// TIA Portal V20 export
FUNCTION_BLOCK "EventsPFE"   // FB183, LAD
// stored: MemoryReserve 100, Namespace Unit1, SetENOAutomatically false
   VAR
      instResourceEvent { S7_SetPoint := 'True'} : "LPFE_ResourceEvent";
      instFEEvent_Taping { S7_SetPoint := 'True'} : "LER_LPFE_FNEvent";
      instFEEvent_HeatPressLeft { S7_SetPoint := 'True'} : "LER_LPFE_FNEvent";
      instFEEvent_HeatPressRight { S7_SetPoint := 'True'} : "LER_LPFE_FNEvent";
      instFEEvent_HipotandThickness { S7_SetPoint := 'True'} : "LER_LPFE_FNEvent";
      instFEEvent_Vision { S7_SetPoint := 'True'} : "LER_LPFE_FNEvent";
      instFEEvent_Laser { S7_SetPoint := 'True'} : "LER_LPFE_FNEvent";
      instFEEvent_Weight { S7_SetPoint := 'True'} : "LER_LPFE_FNEvent";
      InstLPFE_ValueEvent { S7_SetPoint := 'True'} : "LPFE_ValueEvent";
      InstLPFE_TelemetryEventHandlerEM0 { S7_SetPoint := 'True'} : "LPFE_TelemetryEventHandler";
      InstLPFE_TelemetryEventHandlerEM1 { S7_SetPoint := 'True'} : "LPFE_TelemetryEventHandler";
      InstLPFE_TelemetryEventHandlerEM2 { S7_SetPoint := 'True'} : "LPFE_TelemetryEventHandler";
      InstLPFE_TelemetryEventHandlerEM3 { S7_SetPoint := 'True'} : "LPFE_TelemetryEventHandler";
      InstLPFE_TelemetryEventHandlerEM4 { S7_SetPoint := 'True'} : "LPFE_TelemetryEventHandler";
      InstLPFE_TelemetryEventHandlerEM5 { S7_SetPoint := 'True'} : "LPFE_TelemetryEventHandler";
      InstLPFE_TelemetryEventHandlerEM6 { S7_SetPoint := 'True'} : "LPFE_TelemetryEventHandler";
      InstLPFE_TelemetryEventHandlerEM7 { S7_SetPoint := 'True'} : "LPFE_TelemetryEventHandler";
      InstLPFE_TelemetryEventHandlerEM8 { S7_SetPoint := 'True'} : "LPFE_TelemetryEventHandler";
      InstLPFE_TelemetryEventHandlerEM9 { S7_SetPoint := 'True'} : "LPFE_TelemetryEventHandler";
      InstLPFE_TelemetryEventHandlerEM10 { S7_SetPoint := 'True'} : "LPFE_TelemetryEventHandler";
      InstLPFE_TelemetryEventHandlerEM11 { S7_SetPoint := 'True'} : "LPFE_TelemetryEventHandler";
      InstLPFE_TelemetryEventHandlerEM12 { S7_SetPoint := 'True'} : "LPFE_TelemetryEventHandler";
      InstLPFE_TelemetryEventHandlerEM13 { S7_SetPoint := 'True'} : "LPFE_TelemetryEventHandler";
      InstLPFE_RecordEvent { S7_SetPoint := 'True'} : "LPFE_RecordEvent";
   END_VAR
BEGIN

REGION Network 1: Resource Event (4)
   // Configuration example, adpat it according to the event requirements
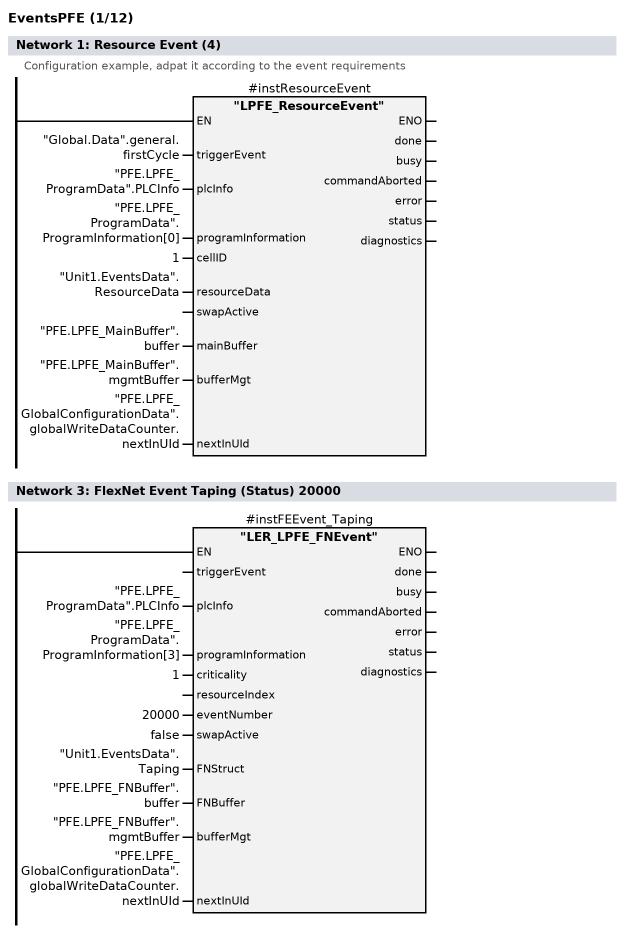
   RUNG wire#powerrail
      #instResourceEvent(triggerEvent := "Global.Data".general.firstCycle, plcInfo := "PFE.LPFE_ProgramData".PLCInfo, programInformation := "PFE.LPFE_ProgramData".ProgramInformation[0], cellID := 1, resourceData := "Unit1.EventsData".ResourceData, swapActive :=, mainBuffer := "PFE.LPFE_MainBuffer".buffer, bufferMgt := "PFE.LPFE_MainBuffer".mgmtBuffer, nextInUId := "PFE.LPFE_GlobalConfigurationData".globalWriteDataCounter.nextInUId, done =>, busy =>, commandAborted =>, error =>, status =>, diagnostics =>)
   END_RUNG
   // the same network as SCL:
   #instResourceEvent(triggerEvent := "Global.Data".general.firstCycle,   // "LPFE_ResourceEvent"
                      plcInfo := "PFE.LPFE_ProgramData".PLCInfo,
                      programInformation := "PFE.LPFE_ProgramData".ProgramInformation[0],
                      cellID := 1,
                      resourceData := "Unit1.EventsData".ResourceData,
                      mainBuffer := "PFE.LPFE_MainBuffer".buffer,
                      bufferMgt := "PFE.LPFE_MainBuffer".mgmtBuffer,
                      nextInUId := "PFE.LPFE_GlobalConfigurationData".globalWriteDataCounter.nextInUId);
END_REGION

REGION Network 3: FlexNet Event Taping (Status) 20000
   RUNG wire#powerrail
      #instFEEvent_Taping(triggerEvent :=, plcInfo := "PFE.LPFE_ProgramData".PLCInfo, programInformation := "PFE.LPFE_ProgramData".ProgramInformation[3], criticality := 1, resourceIndex :=, eventNumber := 20000, swapActive := false, FNStruct := "Unit1.EventsData".Taping, FNBuffer := "PFE.LPFE_FNBuffer".buffer, bufferMgt := "PFE.LPFE_FNBuffer".mgmtBuffer, nextInUId := "PFE.LPFE_GlobalConfigurationData".globalWriteDataCounter.nextInUId, done =>, busy =>, commandAborted =>, error =>, status =>, diagnostics =>)
   END_RUNG
   // the same network as SCL:
   #instFEEvent_Taping(plcInfo := "PFE.LPFE_ProgramData".PLCInfo,   // "LER_LPFE_FNEvent"
                       programInformation := "PFE.LPFE_ProgramData".ProgramInformation[3],
                       criticality := 1,
                       eventNumber := 20000,
                       swapActive := false,
                       FNStruct := "Unit1.EventsData".Taping,
                       FNBuffer := "PFE.LPFE_FNBuffer".buffer,
                       bufferMgt := "PFE.LPFE_FNBuffer".mgmtBuffer,
                       nextInUId := "PFE.LPFE_GlobalConfigurationData".globalWriteDataCounter.nextInUId);
END_REGION

REGION Network 4: FlexNet Event HeatPress - Left (Status) 20001
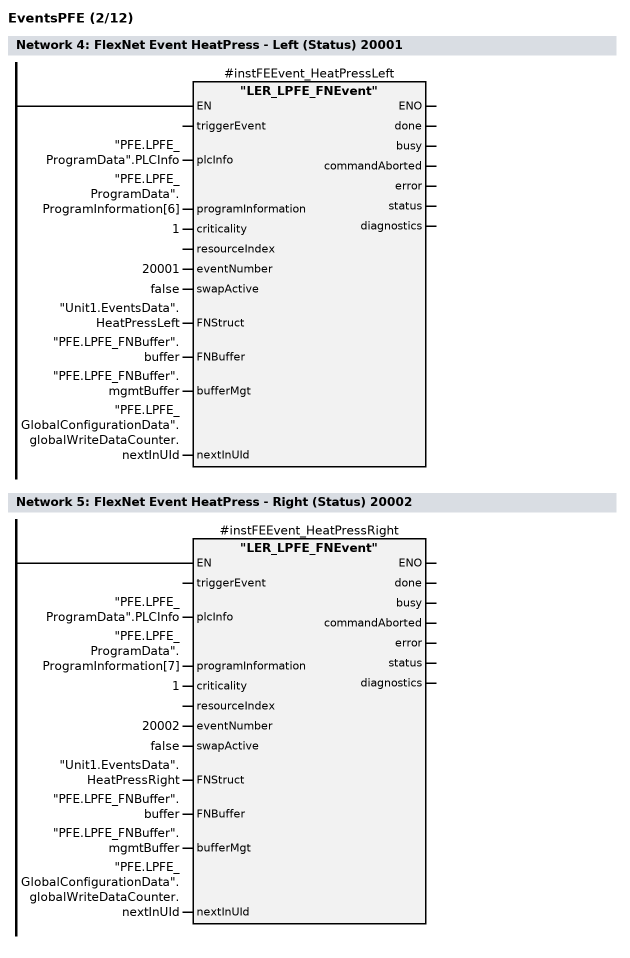
   RUNG wire#powerrail
      #instFEEvent_HeatPressLeft(triggerEvent :=, plcInfo := "PFE.LPFE_ProgramData".PLCInfo, programInformation := "PFE.LPFE_ProgramData".ProgramInformation[6], criticality := 1, resourceIndex :=, eventNumber := 20001, swapActive := false, FNStruct := "Unit1.EventsData".HeatPressLeft, FNBuffer := "PFE.LPFE_FNBuffer".buffer, bufferMgt := "PFE.LPFE_FNBuffer".mgmtBuffer, nextInUId := "PFE.LPFE_GlobalConfigurationData".globalWriteDataCounter.nextInUId, done =>, busy =>, commandAborted =>, error =>, status =>, diagnostics =>)
   END_RUNG
   // the same network as SCL:
   #instFEEvent_HeatPressLeft(plcInfo := "PFE.LPFE_ProgramData".PLCInfo,   // "LER_LPFE_FNEvent"
                           programInformation := "PFE.LPFE_ProgramData".ProgramInformation[6],
                           criticality := 1,
                           eventNumber := 20001,
                           swapActive := false,
                           FNStruct := "Unit1.EventsData".HeatPressLeft,
                           FNBuffer := "PFE.LPFE_FNBuffer".buffer,
                           bufferMgt := "PFE.LPFE_FNBuffer".mgmtBuffer,
                           nextInUId := "PFE.LPFE_GlobalConfigurationData".globalWriteDataCounter.nextInUId);
END_REGION

REGION Network 5: FlexNet Event HeatPress - Right (Status) 20002
   RUNG wire#powerrail
      #instFEEvent_HeatPressRight(triggerEvent :=, plcInfo := "PFE.LPFE_ProgramData".PLCInfo, programInformation := "PFE.LPFE_ProgramData".ProgramInformation[7], criticality := 1, resourceIndex :=, eventNumber := 20002, swapActive := false, FNStruct := "Unit1.EventsData".HeatPressRight, FNBuffer := "PFE.LPFE_FNBuffer".buffer, bufferMgt := "PFE.LPFE_FNBuffer".mgmtBuffer, nextInUId := "PFE.LPFE_GlobalConfigurationData".globalWriteDataCounter.nextInUId, done =>, busy =>, commandAborted =>, error =>, status =>, diagnostics =>)
   END_RUNG
   // the same network as SCL:
   #instFEEvent_HeatPressRight(plcInfo := "PFE.LPFE_ProgramData".PLCInfo,   // "LER_LPFE_FNEvent"
                           programInformation := "PFE.LPFE_ProgramData".ProgramInformation[7],
                           criticality := 1,
                           eventNumber := 20002,
                           swapActive := false,
                           FNStruct := "Unit1.EventsData".HeatPressRight,
                           FNBuffer := "PFE.LPFE_FNBuffer".buffer,
                           bufferMgt := "PFE.LPFE_FNBuffer".mgmtBuffer,
                           nextInUId := "PFE.LPFE_GlobalConfigurationData".globalWriteDataCounter.nextInUId);
END_REGION

REGION Network 6: FlexNet Event Hipot and Thickness (Status) 20003
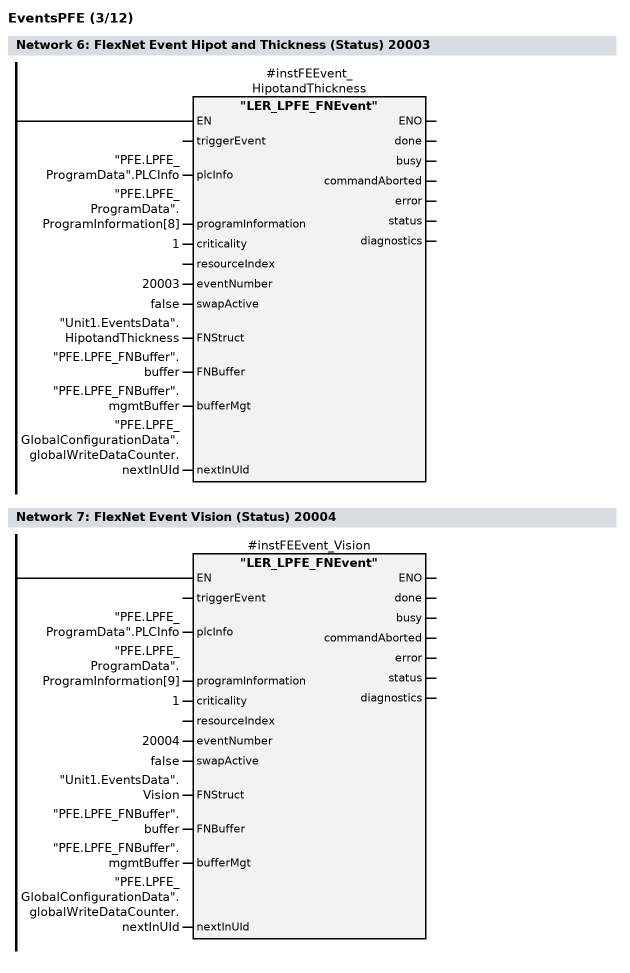
   RUNG wire#powerrail
      #instFEEvent_HipotandThickness(triggerEvent :=, plcInfo := "PFE.LPFE_ProgramData".PLCInfo, programInformation := "PFE.LPFE_ProgramData".ProgramInformation[8], criticality := 1, resourceIndex :=, eventNumber := 20003, swapActive := false, FNStruct := "Unit1.EventsData".HipotandThickness, FNBuffer := "PFE.LPFE_FNBuffer".buffer, bufferMgt := "PFE.LPFE_FNBuffer".mgmtBuffer, nextInUId := "PFE.LPFE_GlobalConfigurationData".globalWriteDataCounter.nextInUId, done =>, busy =>, commandAborted =>, error =>, status =>, diagnostics =>)
   END_RUNG
   // the same network as SCL:
   #instFEEvent_HipotandThickness(plcInfo := "PFE.LPFE_ProgramData".PLCInfo,   // "LER_LPFE_FNEvent"
                           programInformation := "PFE.LPFE_ProgramData".ProgramInformation[8],
                           criticality := 1,
                           eventNumber := 20003,
                           swapActive := false,
                           FNStruct := "Unit1.EventsData".HipotandThickness,
                           FNBuffer := "PFE.LPFE_FNBuffer".buffer,
                           bufferMgt := "PFE.LPFE_FNBuffer".mgmtBuffer,
                           nextInUId := "PFE.LPFE_GlobalConfigurationData".globalWriteDataCounter.nextInUId);
END_REGION

REGION Network 7: FlexNet Event Vision (Status) 20004
   RUNG wire#powerrail
      #instFEEvent_Vision(triggerEvent :=, plcInfo := "PFE.LPFE_ProgramData".PLCInfo, programInformation := "PFE.LPFE_ProgramData".ProgramInformation[9], criticality := 1, resourceIndex :=, eventNumber := 20004, swapActive := false, FNStruct := "Unit1.EventsData".Vision, FNBuffer := "PFE.LPFE_FNBuffer".buffer, bufferMgt := "PFE.LPFE_FNBuffer".mgmtBuffer, nextInUId := "PFE.LPFE_GlobalConfigurationData".globalWriteDataCounter.nextInUId, done =>, busy =>, commandAborted =>, error =>, status =>, diagnostics =>)
   END_RUNG
   // the same network as SCL:
   #instFEEvent_Vision(plcInfo := "PFE.LPFE_ProgramData".PLCInfo,   // "LER_LPFE_FNEvent"
                       programInformation := "PFE.LPFE_ProgramData".ProgramInformation[9],
                       criticality := 1,
                       eventNumber := 20004,
                       swapActive := false,
                       FNStruct := "Unit1.EventsData".Vision,
                       FNBuffer := "PFE.LPFE_FNBuffer".buffer,
                       bufferMgt := "PFE.LPFE_FNBuffer".mgmtBuffer,
                       nextInUId := "PFE.LPFE_GlobalConfigurationData".globalWriteDataCounter.nextInUId);
END_REGION

REGION Network 8: FlexNet Event Laser (Status) 20005
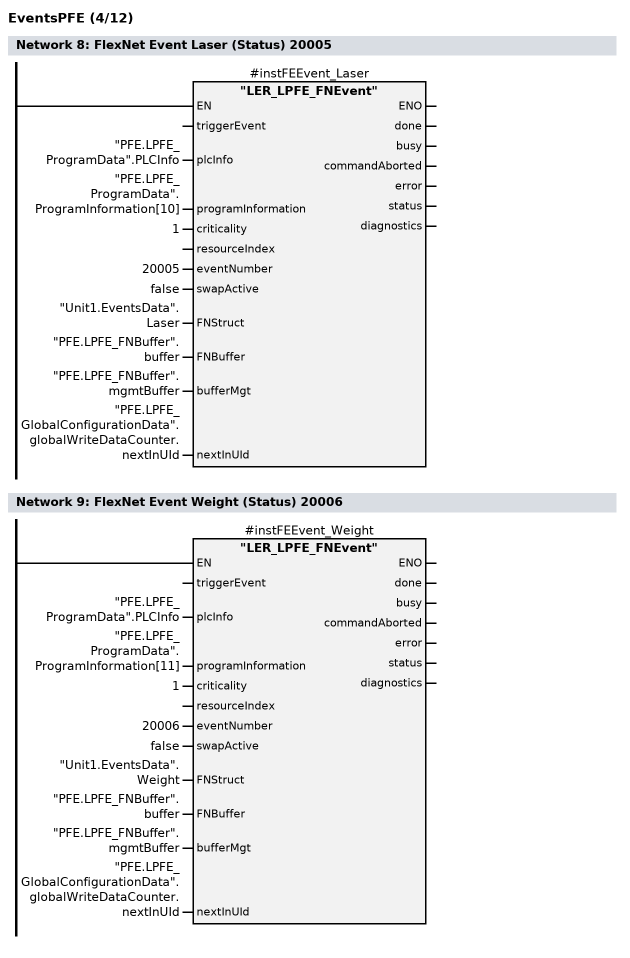
   RUNG wire#powerrail
      #instFEEvent_Laser(triggerEvent :=, plcInfo := "PFE.LPFE_ProgramData".PLCInfo, programInformation := "PFE.LPFE_ProgramData".ProgramInformation[10], criticality := 1, resourceIndex :=, eventNumber := 20005, swapActive := false, FNStruct := "Unit1.EventsData".Laser, FNBuffer := "PFE.LPFE_FNBuffer".buffer, bufferMgt := "PFE.LPFE_FNBuffer".mgmtBuffer, nextInUId := "PFE.LPFE_GlobalConfigurationData".globalWriteDataCounter.nextInUId, done =>, busy =>, commandAborted =>, error =>, status =>, diagnostics =>)
   END_RUNG
   // the same network as SCL:
   #instFEEvent_Laser(plcInfo := "PFE.LPFE_ProgramData".PLCInfo,   // "LER_LPFE_FNEvent"
                      programInformation := "PFE.LPFE_ProgramData".ProgramInformation[10],
                      criticality := 1,
                      eventNumber := 20005,
                      swapActive := false,
                      FNStruct := "Unit1.EventsData".Laser,
                      FNBuffer := "PFE.LPFE_FNBuffer".buffer,
                      bufferMgt := "PFE.LPFE_FNBuffer".mgmtBuffer,
                      nextInUId := "PFE.LPFE_GlobalConfigurationData".globalWriteDataCounter.nextInUId);
END_REGION

REGION Network 9: FlexNet Event Weight (Status) 20006
   RUNG wire#powerrail
      #instFEEvent_Weight(triggerEvent :=, plcInfo := "PFE.LPFE_ProgramData".PLCInfo, programInformation := "PFE.LPFE_ProgramData".ProgramInformation[11], criticality := 1, resourceIndex :=, eventNumber := 20006, swapActive := false, FNStruct := "Unit1.EventsData".Weight, FNBuffer := "PFE.LPFE_FNBuffer".buffer, bufferMgt := "PFE.LPFE_FNBuffer".mgmtBuffer, nextInUId := "PFE.LPFE_GlobalConfigurationData".globalWriteDataCounter.nextInUId, done =>, busy =>, commandAborted =>, error =>, status =>, diagnostics =>)
   END_RUNG
   // the same network as SCL:
   #instFEEvent_Weight(plcInfo := "PFE.LPFE_ProgramData".PLCInfo,   // "LER_LPFE_FNEvent"
                       programInformation := "PFE.LPFE_ProgramData".ProgramInformation[11],
                       criticality := 1,
                       eventNumber := 20006,
                       swapActive := false,
                       FNStruct := "Unit1.EventsData".Weight,
                       FNBuffer := "PFE.LPFE_FNBuffer".buffer,
                       bufferMgt := "PFE.LPFE_FNBuffer".mgmtBuffer,
                       nextInUId := "PFE.LPFE_GlobalConfigurationData".globalWriteDataCounter.nextInUId);
END_REGION

REGION Network 10: ValueEvent (6)
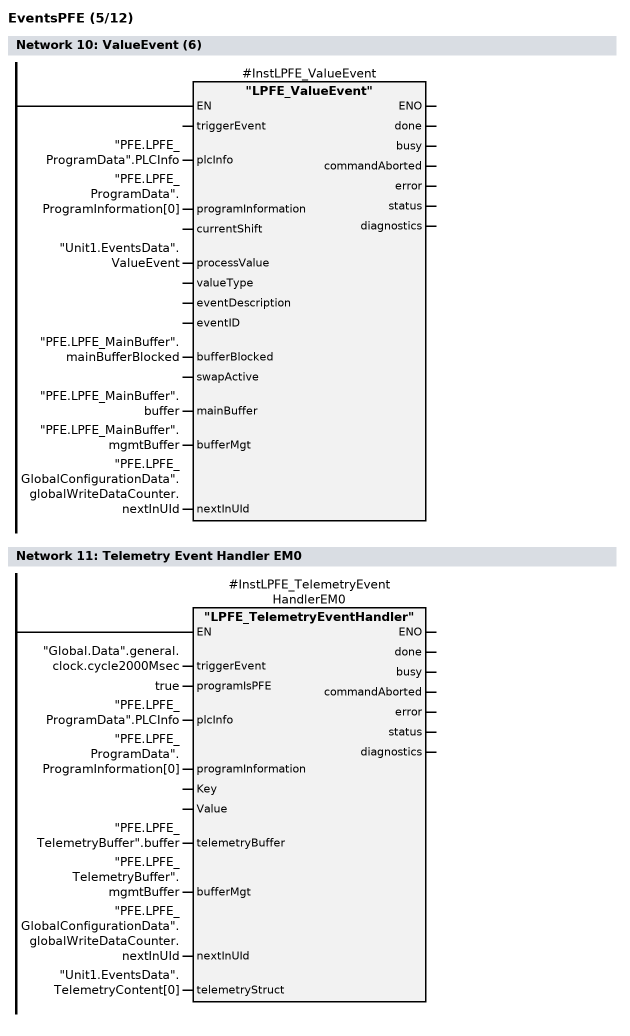
   RUNG wire#powerrail
      #InstLPFE_ValueEvent(triggerEvent :=, plcInfo := "PFE.LPFE_ProgramData".PLCInfo, programInformation := "PFE.LPFE_ProgramData".ProgramInformation[0], currentShift :=, processValue := "Unit1.EventsData".ValueEvent, valueType :=, eventDescription :=, eventID :=, bufferBlocked := "PFE.LPFE_MainBuffer".mainBufferBlocked, swapActive :=, mainBuffer := "PFE.LPFE_MainBuffer".buffer, bufferMgt := "PFE.LPFE_MainBuffer".mgmtBuffer, nextInUId := "PFE.LPFE_GlobalConfigurationData".globalWriteDataCounter.nextInUId, done =>, busy =>, commandAborted =>, error =>, status =>, diagnostics =>)
   END_RUNG
   // the same network as SCL:
   #InstLPFE_ValueEvent(plcInfo := "PFE.LPFE_ProgramData".PLCInfo,   // "LPFE_ValueEvent"
                        programInformation := "PFE.LPFE_ProgramData".ProgramInformation[0],
                        processValue := "Unit1.EventsData".ValueEvent,
                        bufferBlocked := "PFE.LPFE_MainBuffer".mainBufferBlocked,
                        mainBuffer := "PFE.LPFE_MainBuffer".buffer,
                        bufferMgt := "PFE.LPFE_MainBuffer".mgmtBuffer,
                        nextInUId := "PFE.LPFE_GlobalConfigurationData".globalWriteDataCounter.nextInUId);
END_REGION

REGION Network 11: Telemetry Event Handler EM0
   RUNG wire#powerrail
      #InstLPFE_TelemetryEventHandlerEM0(triggerEvent := "Global.Data".general.clock.cycle2000Msec, programIsPFE := true, plcInfo := "PFE.LPFE_ProgramData".PLCInfo, programInformation := "PFE.LPFE_ProgramData".ProgramInformation[0], Key :=, Value :=, telemetryBuffer := "PFE.LPFE_TelemetryBuffer".buffer, bufferMgt := "PFE.LPFE_TelemetryBuffer".mgmtBuffer, nextInUId := "PFE.LPFE_GlobalConfigurationData".globalWriteDataCounter.nextInUId, telemetryStruct := "Unit1.EventsData".TelemetryContent[0], done =>, busy =>, commandAborted =>, error =>, status =>, diagnostics =>)
   END_RUNG
   // the same network as SCL:
   #InstLPFE_TelemetryEventHandlerEM0(triggerEvent := "Global.Data".general.clock.cycle2000Msec,   // "LPFE_TelemetryEventHandler"
                           programIsPFE := true,
                           plcInfo := "PFE.LPFE_ProgramData".PLCInfo,
                           programInformation := "PFE.LPFE_ProgramData".ProgramInformation[0],
                           telemetryBuffer := "PFE.LPFE_TelemetryBuffer".buffer,
                           bufferMgt := "PFE.LPFE_TelemetryBuffer".mgmtBuffer,
                           nextInUId := "PFE.LPFE_GlobalConfigurationData".globalWriteDataCounter.nextInUId,
                           telemetryStruct := "Unit1.EventsData".TelemetryContent[0]);
END_REGION

REGION Network 12: Telemetry Event Handler EM1
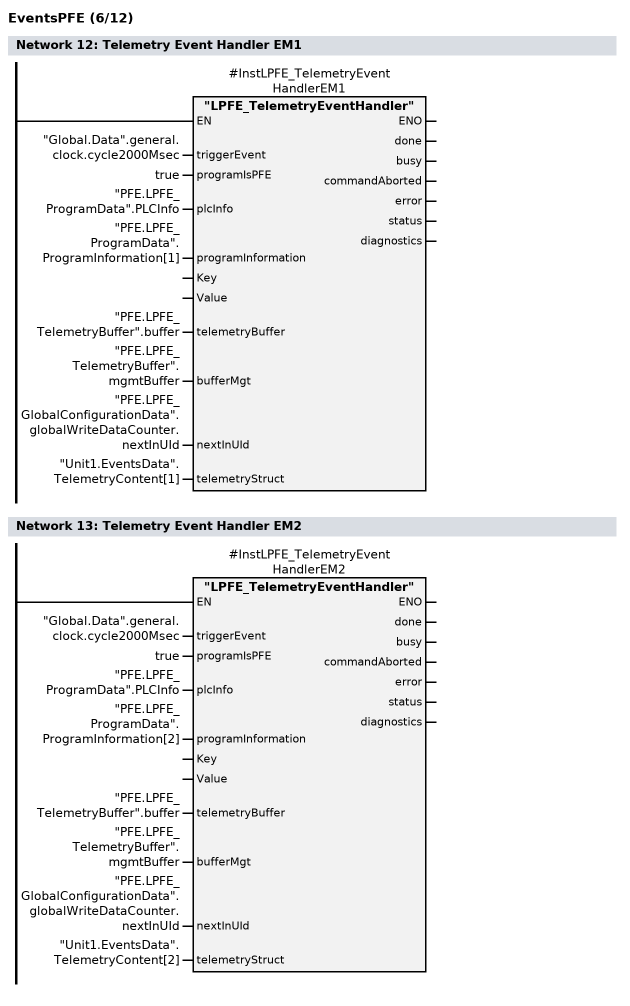
   RUNG wire#powerrail
      #InstLPFE_TelemetryEventHandlerEM1(triggerEvent := "Global.Data".general.clock.cycle2000Msec, programIsPFE := true, plcInfo := "PFE.LPFE_ProgramData".PLCInfo, programInformation := "PFE.LPFE_ProgramData".ProgramInformation[1], Key :=, Value :=, telemetryBuffer := "PFE.LPFE_TelemetryBuffer".buffer, bufferMgt := "PFE.LPFE_TelemetryBuffer".mgmtBuffer, nextInUId := "PFE.LPFE_GlobalConfigurationData".globalWriteDataCounter.nextInUId, telemetryStruct := "Unit1.EventsData".TelemetryContent[1], done =>, busy =>, commandAborted =>, error =>, status =>, diagnostics =>)
   END_RUNG
   // the same network as SCL:
   #InstLPFE_TelemetryEventHandlerEM1(triggerEvent := "Global.Data".general.clock.cycle2000Msec,   // "LPFE_TelemetryEventHandler"
                           programIsPFE := true,
                           plcInfo := "PFE.LPFE_ProgramData".PLCInfo,
                           programInformation := "PFE.LPFE_ProgramData".ProgramInformation[1],
                           telemetryBuffer := "PFE.LPFE_TelemetryBuffer".buffer,
                           bufferMgt := "PFE.LPFE_TelemetryBuffer".mgmtBuffer,
                           nextInUId := "PFE.LPFE_GlobalConfigurationData".globalWriteDataCounter.nextInUId,
                           telemetryStruct := "Unit1.EventsData".TelemetryContent[1]);
END_REGION

REGION Network 13: Telemetry Event Handler EM2
   RUNG wire#powerrail
      #InstLPFE_TelemetryEventHandlerEM2(triggerEvent := "Global.Data".general.clock.cycle2000Msec, programIsPFE := true, plcInfo := "PFE.LPFE_ProgramData".PLCInfo, programInformation := "PFE.LPFE_ProgramData".ProgramInformation[2], Key :=, Value :=, telemetryBuffer := "PFE.LPFE_TelemetryBuffer".buffer, bufferMgt := "PFE.LPFE_TelemetryBuffer".mgmtBuffer, nextInUId := "PFE.LPFE_GlobalConfigurationData".globalWriteDataCounter.nextInUId, telemetryStruct := "Unit1.EventsData".TelemetryContent[2], done =>, busy =>, commandAborted =>, error =>, status =>, diagnostics =>)
   END_RUNG
   // the same network as SCL:
   #InstLPFE_TelemetryEventHandlerEM2(triggerEvent := "Global.Data".general.clock.cycle2000Msec,   // "LPFE_TelemetryEventHandler"
                           programIsPFE := true,
                           plcInfo := "PFE.LPFE_ProgramData".PLCInfo,
                           programInformation := "PFE.LPFE_ProgramData".ProgramInformation[2],
                           telemetryBuffer := "PFE.LPFE_TelemetryBuffer".buffer,
                           bufferMgt := "PFE.LPFE_TelemetryBuffer".mgmtBuffer,
                           nextInUId := "PFE.LPFE_GlobalConfigurationData".globalWriteDataCounter.nextInUId,
                           telemetryStruct := "Unit1.EventsData".TelemetryContent[2]);
END_REGION

REGION Network 14: Telemetry Event Handler EM3
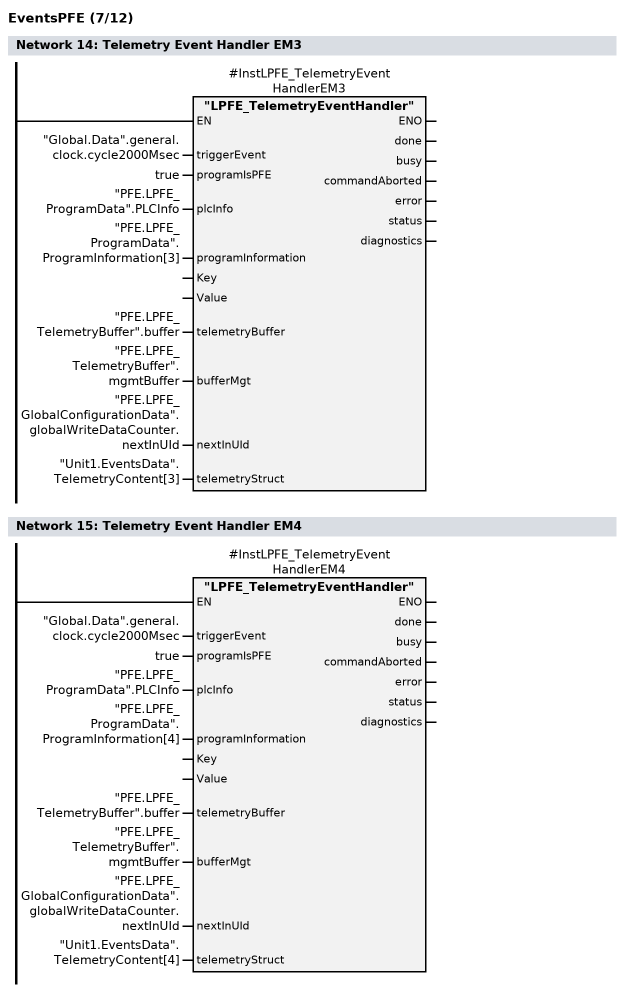
   RUNG wire#powerrail
      #InstLPFE_TelemetryEventHandlerEM3(triggerEvent := "Global.Data".general.clock.cycle2000Msec, programIsPFE := true, plcInfo := "PFE.LPFE_ProgramData".PLCInfo, programInformation := "PFE.LPFE_ProgramData".ProgramInformation[3], Key :=, Value :=, telemetryBuffer := "PFE.LPFE_TelemetryBuffer".buffer, bufferMgt := "PFE.LPFE_TelemetryBuffer".mgmtBuffer, nextInUId := "PFE.LPFE_GlobalConfigurationData".globalWriteDataCounter.nextInUId, telemetryStruct := "Unit1.EventsData".TelemetryContent[3], done =>, busy =>, commandAborted =>, error =>, status =>, diagnostics =>)
   END_RUNG
   // the same network as SCL:
   #InstLPFE_TelemetryEventHandlerEM3(triggerEvent := "Global.Data".general.clock.cycle2000Msec,   // "LPFE_TelemetryEventHandler"
                           programIsPFE := true,
                           plcInfo := "PFE.LPFE_ProgramData".PLCInfo,
                           programInformation := "PFE.LPFE_ProgramData".ProgramInformation[3],
                           telemetryBuffer := "PFE.LPFE_TelemetryBuffer".buffer,
                           bufferMgt := "PFE.LPFE_TelemetryBuffer".mgmtBuffer,
                           nextInUId := "PFE.LPFE_GlobalConfigurationData".globalWriteDataCounter.nextInUId,
                           telemetryStruct := "Unit1.EventsData".TelemetryContent[3]);
END_REGION

REGION Network 15: Telemetry Event Handler EM4
   RUNG wire#powerrail
      #InstLPFE_TelemetryEventHandlerEM4(triggerEvent := "Global.Data".general.clock.cycle2000Msec, programIsPFE := true, plcInfo := "PFE.LPFE_ProgramData".PLCInfo, programInformation := "PFE.LPFE_ProgramData".ProgramInformation[4], Key :=, Value :=, telemetryBuffer := "PFE.LPFE_TelemetryBuffer".buffer, bufferMgt := "PFE.LPFE_TelemetryBuffer".mgmtBuffer, nextInUId := "PFE.LPFE_GlobalConfigurationData".globalWriteDataCounter.nextInUId, telemetryStruct := "Unit1.EventsData".TelemetryContent[4], done =>, busy =>, commandAborted =>, error =>, status =>, diagnostics =>)
   END_RUNG
   // the same network as SCL:
   #InstLPFE_TelemetryEventHandlerEM4(triggerEvent := "Global.Data".general.clock.cycle2000Msec,   // "LPFE_TelemetryEventHandler"
                           programIsPFE := true,
                           plcInfo := "PFE.LPFE_ProgramData".PLCInfo,
                           programInformation := "PFE.LPFE_ProgramData".ProgramInformation[4],
                           telemetryBuffer := "PFE.LPFE_TelemetryBuffer".buffer,
                           bufferMgt := "PFE.LPFE_TelemetryBuffer".mgmtBuffer,
                           nextInUId := "PFE.LPFE_GlobalConfigurationData".globalWriteDataCounter.nextInUId,
                           telemetryStruct := "Unit1.EventsData".TelemetryContent[4]);
END_REGION

REGION Network 16: Telemetry Event Handler EM5
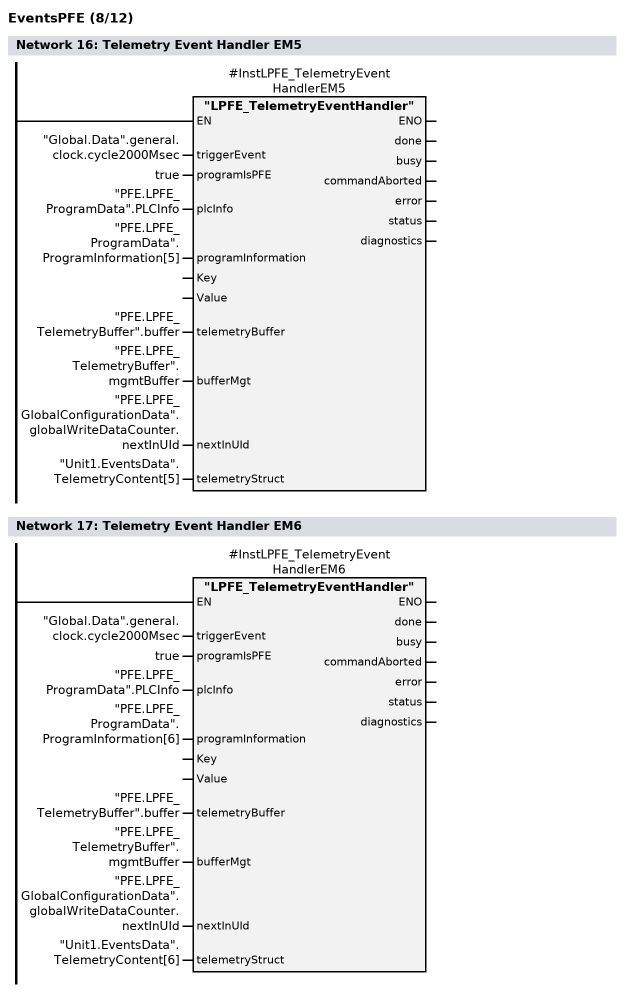
   RUNG wire#powerrail
      #InstLPFE_TelemetryEventHandlerEM5(triggerEvent := "Global.Data".general.clock.cycle2000Msec, programIsPFE := true, plcInfo := "PFE.LPFE_ProgramData".PLCInfo, programInformation := "PFE.LPFE_ProgramData".ProgramInformation[5], Key :=, Value :=, telemetryBuffer := "PFE.LPFE_TelemetryBuffer".buffer, bufferMgt := "PFE.LPFE_TelemetryBuffer".mgmtBuffer, nextInUId := "PFE.LPFE_GlobalConfigurationData".globalWriteDataCounter.nextInUId, telemetryStruct := "Unit1.EventsData".TelemetryContent[5], done =>, busy =>, commandAborted =>, error =>, status =>, diagnostics =>)
   END_RUNG
   // the same network as SCL:
   #InstLPFE_TelemetryEventHandlerEM5(triggerEvent := "Global.Data".general.clock.cycle2000Msec,   // "LPFE_TelemetryEventHandler"
                           programIsPFE := true,
                           plcInfo := "PFE.LPFE_ProgramData".PLCInfo,
                           programInformation := "PFE.LPFE_ProgramData".ProgramInformation[5],
                           telemetryBuffer := "PFE.LPFE_TelemetryBuffer".buffer,
                           bufferMgt := "PFE.LPFE_TelemetryBuffer".mgmtBuffer,
                           nextInUId := "PFE.LPFE_GlobalConfigurationData".globalWriteDataCounter.nextInUId,
                           telemetryStruct := "Unit1.EventsData".TelemetryContent[5]);
END_REGION

REGION Network 17: Telemetry Event Handler EM6
   RUNG wire#powerrail
      #InstLPFE_TelemetryEventHandlerEM6(triggerEvent := "Global.Data".general.clock.cycle2000Msec, programIsPFE := true, plcInfo := "PFE.LPFE_ProgramData".PLCInfo, programInformation := "PFE.LPFE_ProgramData".ProgramInformation[6], Key :=, Value :=, telemetryBuffer := "PFE.LPFE_TelemetryBuffer".buffer, bufferMgt := "PFE.LPFE_TelemetryBuffer".mgmtBuffer, nextInUId := "PFE.LPFE_GlobalConfigurationData".globalWriteDataCounter.nextInUId, telemetryStruct := "Unit1.EventsData".TelemetryContent[6], done =>, busy =>, commandAborted =>, error =>, status =>, diagnostics =>)
   END_RUNG
   // the same network as SCL:
   #InstLPFE_TelemetryEventHandlerEM6(triggerEvent := "Global.Data".general.clock.cycle2000Msec,   // "LPFE_TelemetryEventHandler"
                           programIsPFE := true,
                           plcInfo := "PFE.LPFE_ProgramData".PLCInfo,
                           programInformation := "PFE.LPFE_ProgramData".ProgramInformation[6],
                           telemetryBuffer := "PFE.LPFE_TelemetryBuffer".buffer,
                           bufferMgt := "PFE.LPFE_TelemetryBuffer".mgmtBuffer,
                           nextInUId := "PFE.LPFE_GlobalConfigurationData".globalWriteDataCounter.nextInUId,
                           telemetryStruct := "Unit1.EventsData".TelemetryContent[6]);
END_REGION

REGION Network 18: Telemetry Event Handler EM7
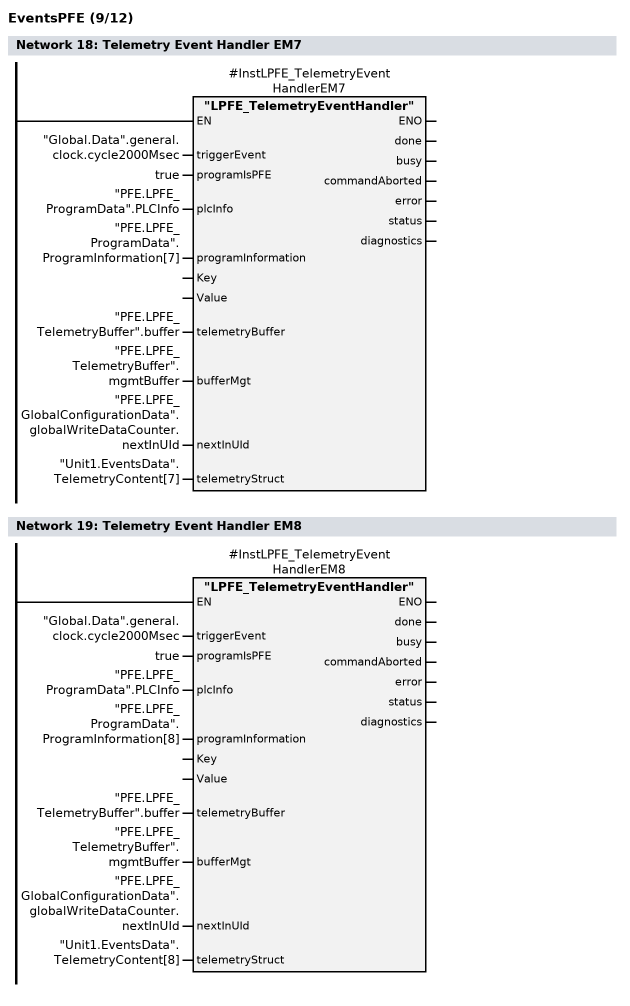
   RUNG wire#powerrail
      #InstLPFE_TelemetryEventHandlerEM7(triggerEvent := "Global.Data".general.clock.cycle2000Msec, programIsPFE := true, plcInfo := "PFE.LPFE_ProgramData".PLCInfo, programInformation := "PFE.LPFE_ProgramData".ProgramInformation[7], Key :=, Value :=, telemetryBuffer := "PFE.LPFE_TelemetryBuffer".buffer, bufferMgt := "PFE.LPFE_TelemetryBuffer".mgmtBuffer, nextInUId := "PFE.LPFE_GlobalConfigurationData".globalWriteDataCounter.nextInUId, telemetryStruct := "Unit1.EventsData".TelemetryContent[7], done =>, busy =>, commandAborted =>, error =>, status =>, diagnostics =>)
   END_RUNG
   // the same network as SCL:
   #InstLPFE_TelemetryEventHandlerEM7(triggerEvent := "Global.Data".general.clock.cycle2000Msec,   // "LPFE_TelemetryEventHandler"
                           programIsPFE := true,
                           plcInfo := "PFE.LPFE_ProgramData".PLCInfo,
                           programInformation := "PFE.LPFE_ProgramData".ProgramInformation[7],
                           telemetryBuffer := "PFE.LPFE_TelemetryBuffer".buffer,
                           bufferMgt := "PFE.LPFE_TelemetryBuffer".mgmtBuffer,
                           nextInUId := "PFE.LPFE_GlobalConfigurationData".globalWriteDataCounter.nextInUId,
                           telemetryStruct := "Unit1.EventsData".TelemetryContent[7]);
END_REGION

REGION Network 19: Telemetry Event Handler EM8
   RUNG wire#powerrail
      #InstLPFE_TelemetryEventHandlerEM8(triggerEvent := "Global.Data".general.clock.cycle2000Msec, programIsPFE := true, plcInfo := "PFE.LPFE_ProgramData".PLCInfo, programInformation := "PFE.LPFE_ProgramData".ProgramInformation[8], Key :=, Value :=, telemetryBuffer := "PFE.LPFE_TelemetryBuffer".buffer, bufferMgt := "PFE.LPFE_TelemetryBuffer".mgmtBuffer, nextInUId := "PFE.LPFE_GlobalConfigurationData".globalWriteDataCounter.nextInUId, telemetryStruct := "Unit1.EventsData".TelemetryContent[8], done =>, busy =>, commandAborted =>, error =>, status =>, diagnostics =>)
   END_RUNG
   // the same network as SCL:
   #InstLPFE_TelemetryEventHandlerEM8(triggerEvent := "Global.Data".general.clock.cycle2000Msec,   // "LPFE_TelemetryEventHandler"
                           programIsPFE := true,
                           plcInfo := "PFE.LPFE_ProgramData".PLCInfo,
                           programInformation := "PFE.LPFE_ProgramData".ProgramInformation[8],
                           telemetryBuffer := "PFE.LPFE_TelemetryBuffer".buffer,
                           bufferMgt := "PFE.LPFE_TelemetryBuffer".mgmtBuffer,
                           nextInUId := "PFE.LPFE_GlobalConfigurationData".globalWriteDataCounter.nextInUId,
                           telemetryStruct := "Unit1.EventsData".TelemetryContent[8]);
END_REGION

REGION Network 20: Telemetry Event Handler EM9
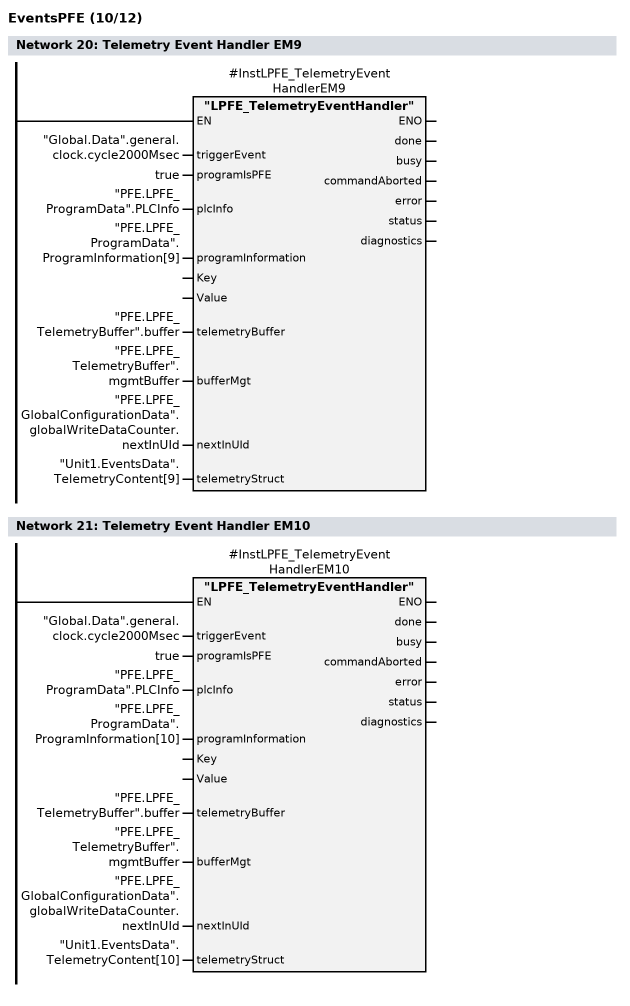
   RUNG wire#powerrail
      #InstLPFE_TelemetryEventHandlerEM9(triggerEvent := "Global.Data".general.clock.cycle2000Msec, programIsPFE := true, plcInfo := "PFE.LPFE_ProgramData".PLCInfo, programInformation := "PFE.LPFE_ProgramData".ProgramInformation[9], Key :=, Value :=, telemetryBuffer := "PFE.LPFE_TelemetryBuffer".buffer, bufferMgt := "PFE.LPFE_TelemetryBuffer".mgmtBuffer, nextInUId := "PFE.LPFE_GlobalConfigurationData".globalWriteDataCounter.nextInUId, telemetryStruct := "Unit1.EventsData".TelemetryContent[9], done =>, busy =>, commandAborted =>, error =>, status =>, diagnostics =>)
   END_RUNG
   // the same network as SCL:
   #InstLPFE_TelemetryEventHandlerEM9(triggerEvent := "Global.Data".general.clock.cycle2000Msec,   // "LPFE_TelemetryEventHandler"
                           programIsPFE := true,
                           plcInfo := "PFE.LPFE_ProgramData".PLCInfo,
                           programInformation := "PFE.LPFE_ProgramData".ProgramInformation[9],
                           telemetryBuffer := "PFE.LPFE_TelemetryBuffer".buffer,
                           bufferMgt := "PFE.LPFE_TelemetryBuffer".mgmtBuffer,
                           nextInUId := "PFE.LPFE_GlobalConfigurationData".globalWriteDataCounter.nextInUId,
                           telemetryStruct := "Unit1.EventsData".TelemetryContent[9]);
END_REGION

REGION Network 21: Telemetry Event Handler EM10
   RUNG wire#powerrail
      #InstLPFE_TelemetryEventHandlerEM10(triggerEvent := "Global.Data".general.clock.cycle2000Msec, programIsPFE := true, plcInfo := "PFE.LPFE_ProgramData".PLCInfo, programInformation := "PFE.LPFE_ProgramData".ProgramInformation[10], Key :=, Value :=, telemetryBuffer := "PFE.LPFE_TelemetryBuffer".buffer, bufferMgt := "PFE.LPFE_TelemetryBuffer".mgmtBuffer, nextInUId := "PFE.LPFE_GlobalConfigurationData".globalWriteDataCounter.nextInUId, telemetryStruct := "Unit1.EventsData".TelemetryContent[10], done =>, busy =>, commandAborted =>, error =>, status =>, diagnostics =>)
   END_RUNG
   // the same network as SCL:
   #InstLPFE_TelemetryEventHandlerEM10(triggerEvent := "Global.Data".general.clock.cycle2000Msec,   // "LPFE_TelemetryEventHandler"
                           programIsPFE := true,
                           plcInfo := "PFE.LPFE_ProgramData".PLCInfo,
                           programInformation := "PFE.LPFE_ProgramData".ProgramInformation[10],
                           telemetryBuffer := "PFE.LPFE_TelemetryBuffer".buffer,
                           bufferMgt := "PFE.LPFE_TelemetryBuffer".mgmtBuffer,
                           nextInUId := "PFE.LPFE_GlobalConfigurationData".globalWriteDataCounter.nextInUId,
                           telemetryStruct := "Unit1.EventsData".TelemetryContent[10]);
END_REGION

REGION Network 22: Telemetry Event Handler EM11
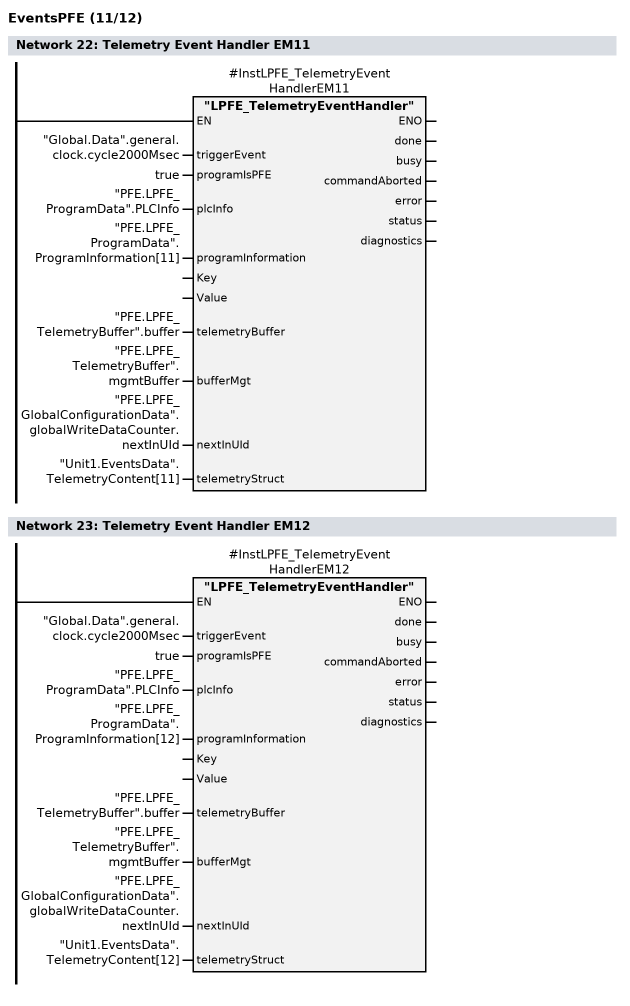
   RUNG wire#powerrail
      #InstLPFE_TelemetryEventHandlerEM11(triggerEvent := "Global.Data".general.clock.cycle2000Msec, programIsPFE := true, plcInfo := "PFE.LPFE_ProgramData".PLCInfo, programInformation := "PFE.LPFE_ProgramData".ProgramInformation[11], Key :=, Value :=, telemetryBuffer := "PFE.LPFE_TelemetryBuffer".buffer, bufferMgt := "PFE.LPFE_TelemetryBuffer".mgmtBuffer, nextInUId := "PFE.LPFE_GlobalConfigurationData".globalWriteDataCounter.nextInUId, telemetryStruct := "Unit1.EventsData".TelemetryContent[11], done =>, busy =>, commandAborted =>, error =>, status =>, diagnostics =>)
   END_RUNG
   // the same network as SCL:
   #InstLPFE_TelemetryEventHandlerEM11(triggerEvent := "Global.Data".general.clock.cycle2000Msec,   // "LPFE_TelemetryEventHandler"
                           programIsPFE := true,
                           plcInfo := "PFE.LPFE_ProgramData".PLCInfo,
                           programInformation := "PFE.LPFE_ProgramData".ProgramInformation[11],
                           telemetryBuffer := "PFE.LPFE_TelemetryBuffer".buffer,
                           bufferMgt := "PFE.LPFE_TelemetryBuffer".mgmtBuffer,
                           nextInUId := "PFE.LPFE_GlobalConfigurationData".globalWriteDataCounter.nextInUId,
                           telemetryStruct := "Unit1.EventsData".TelemetryContent[11]);
END_REGION

REGION Network 23: Telemetry Event Handler EM12
   RUNG wire#powerrail
      #InstLPFE_TelemetryEventHandlerEM12(triggerEvent := "Global.Data".general.clock.cycle2000Msec, programIsPFE := true, plcInfo := "PFE.LPFE_ProgramData".PLCInfo, programInformation := "PFE.LPFE_ProgramData".ProgramInformation[12], Key :=, Value :=, telemetryBuffer := "PFE.LPFE_TelemetryBuffer".buffer, bufferMgt := "PFE.LPFE_TelemetryBuffer".mgmtBuffer, nextInUId := "PFE.LPFE_GlobalConfigurationData".globalWriteDataCounter.nextInUId, telemetryStruct := "Unit1.EventsData".TelemetryContent[12], done =>, busy =>, commandAborted =>, error =>, status =>, diagnostics =>)
   END_RUNG
   // the same network as SCL:
   #InstLPFE_TelemetryEventHandlerEM12(triggerEvent := "Global.Data".general.clock.cycle2000Msec,   // "LPFE_TelemetryEventHandler"
                           programIsPFE := true,
                           plcInfo := "PFE.LPFE_ProgramData".PLCInfo,
                           programInformation := "PFE.LPFE_ProgramData".ProgramInformation[12],
                           telemetryBuffer := "PFE.LPFE_TelemetryBuffer".buffer,
                           bufferMgt := "PFE.LPFE_TelemetryBuffer".mgmtBuffer,
                           nextInUId := "PFE.LPFE_GlobalConfigurationData".globalWriteDataCounter.nextInUId,
                           telemetryStruct := "Unit1.EventsData".TelemetryContent[12]);
END_REGION

REGION Network 24: Telemetry Event Handler EM13
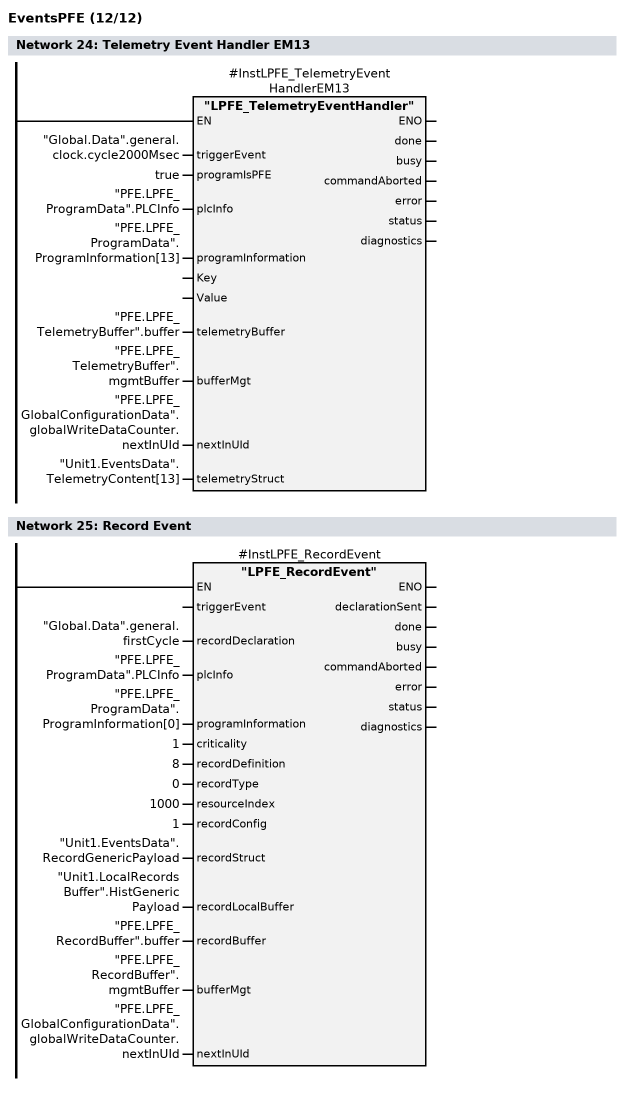
   RUNG wire#powerrail
      #InstLPFE_TelemetryEventHandlerEM13(triggerEvent := "Global.Data".general.clock.cycle2000Msec, programIsPFE := true, plcInfo := "PFE.LPFE_ProgramData".PLCInfo, programInformation := "PFE.LPFE_ProgramData".ProgramInformation[13], Key :=, Value :=, telemetryBuffer := "PFE.LPFE_TelemetryBuffer".buffer, bufferMgt := "PFE.LPFE_TelemetryBuffer".mgmtBuffer, nextInUId := "PFE.LPFE_GlobalConfigurationData".globalWriteDataCounter.nextInUId, telemetryStruct := "Unit1.EventsData".TelemetryContent[13], done =>, busy =>, commandAborted =>, error =>, status =>, diagnostics =>)
   END_RUNG
   // the same network as SCL:
   #InstLPFE_TelemetryEventHandlerEM13(triggerEvent := "Global.Data".general.clock.cycle2000Msec,   // "LPFE_TelemetryEventHandler"
                           programIsPFE := true,
                           plcInfo := "PFE.LPFE_ProgramData".PLCInfo,
                           programInformation := "PFE.LPFE_ProgramData".ProgramInformation[13],
                           telemetryBuffer := "PFE.LPFE_TelemetryBuffer".buffer,
                           bufferMgt := "PFE.LPFE_TelemetryBuffer".mgmtBuffer,
                           nextInUId := "PFE.LPFE_GlobalConfigurationData".globalWriteDataCounter.nextInUId,
                           telemetryStruct := "Unit1.EventsData".TelemetryContent[13]);
END_REGION

REGION Network 25: Record Event
   RUNG wire#powerrail
      #InstLPFE_RecordEvent(triggerEvent :=, recordDeclaration := "Global.Data".general.firstCycle, plcInfo := "PFE.LPFE_ProgramData".PLCInfo, programInformation := "PFE.LPFE_ProgramData".ProgramInformation[0], criticality := 1, recordDefinition := 8, recordType := 0, resourceIndex := 1000, recordConfig := 1, recordStruct := "Unit1.EventsData".RecordGenericPayload, recordLocalBuffer := "Unit1.LocalRecordsBuffer".HistGenericPayload, recordBuffer := "PFE.LPFE_RecordBuffer".buffer, bufferMgt := "PFE.LPFE_RecordBuffer".mgmtBuffer, nextInUId := "PFE.LPFE_GlobalConfigurationData".globalWriteDataCounter.nextInUId, declarationSent =>, done =>, busy =>, commandAborted =>, error =>, status =>, diagnostics =>)
   END_RUNG
   // the same network as SCL:
   #InstLPFE_RecordEvent(recordDeclaration := "Global.Data".general.firstCycle,   // "LPFE_RecordEvent"
                         plcInfo := "PFE.LPFE_ProgramData".PLCInfo,
                         programInformation := "PFE.LPFE_ProgramData".ProgramInformation[0],
                         criticality := 1,
                         recordDefinition := 8,
                         recordType := 0,
                         resourceIndex := 1000,
                         recordConfig := 1,
                         recordStruct := "Unit1.EventsData".RecordGenericPayload,
                         recordLocalBuffer := "Unit1.LocalRecordsBuffer".HistGenericPayload,
                         recordBuffer := "PFE.LPFE_RecordBuffer".buffer,
                         bufferMgt := "PFE.LPFE_RecordBuffer".mgmtBuffer,
                         nextInUId := "PFE.LPFE_GlobalConfigurationData".globalWriteDataCounter.nextInUId);
END_REGION

REGION Network 26: End of the Structure
END_REGION
END_FUNCTION_BLOCK
